// TIA Portal project "SiemensS7-modbus-TCPIP-server" (V16)

(* hardware
DEVICE "S71500/ET200MP station_1"  S7-1500 station
   slot 0: "Rail_0"  Rack  6ES7 590-1***0-0AA0
   slot 1: "PLC_1"  CPU 1512C-1 PN  6ES7 512-1CK01-0AB0  V2.8
      slot 3: "CPU display_1"  6ES7591-1AA00-0AA0
      slot 32768: "PROFINET interface_1"  X1
         slot 32769: "Port_1"  X1 P1
         slot 32770: "Port_2"  X1 P2
      slot 34817: "Virtual CP interface port_1"  Virtual CP interface port  Virtual CP interface port
*)

// ===== PLC "PLC_1"  CPU 1512C-1 PN =====

VAR_GLOBAL   // PLC tag table "Default tag table"
   "System_Byte" AT %MB1 : Byte;
   "FirstScan" AT %M1.0 : Bool;
   "DiagStatusUpdate" AT %M1.1 : Bool;
   "AlwaysTRUE" AT %M1.2 : Bool;
   "AlwaysFALSE" AT %M1.3 : Bool;
   "Clock_Byte" AT %MB0 : Byte;
   "Clock_10Hz" AT %M0.0 : Bool;
   "Clock_5Hz" AT %M0.1 : Bool;
   "Clock_2.5Hz" AT %M0.2 : Bool;
   "Clock_2Hz" AT %M0.3 : Bool;
   "Clock_1.25Hz" AT %M0.4 : Bool;
   "Clock_1Hz" AT %M0.5 : Bool;
   "Clock_0.625Hz" AT %M0.6 : Bool;
   "Clock_0.5Hz" AT %M0.7 : Bool;
   "Tag_1" AT %M1.4 : Bool;
END_VAR

DATA_BLOCK "Connect"   // DB1
{ S7_Optimized_Access := 'FALSE' }
VERSION : 0.1
   VAR
      Req : Bool := false;
      Disconnect : Bool;
      SND : TCON_IP_v4;
      RCV : TCON_IP_v4;
   END_VAR
BEGIN
   SND.InterfaceId := 64;
   SND.ID := 1;
   SND.ConnectionType := 11;
   SND.ActiveEstablished := True;
   SND.RemotePort := 502;
   SND.RemoteAddress.ADDR[1] := 192;
   SND.RemoteAddress.ADDR[2] := 168;
   SND.RemoteAddress.ADDR[3] := 0;
   SND.RemoteAddress.ADDR[4] := 114;
   RCV.InterfaceId := 64;
   RCV.ID := 2;
   RCV.ConnectionType := 11;
   RCV.ActiveEstablished := True;
   RCV.RemoteAddress.ADDR[1] := 192;
   RCV.RemoteAddress.ADDR[2] := 168;
   RCV.RemoteAddress.ADDR[3] := 0;
   RCV.RemoteAddress.ADDR[4] := 114;
   RCV.RemotePort := 502;
   SND.LocalPort := 0;
   RCV.LocalPort := 0;
END_DATA_BLOCK

DATA_BLOCK "Data"   // DB2
{ S7_Optimized_Access := 'FALSE' }
VERSION : 0.1
   VAR
      SND : Array[0..3] of Int;
      RCV : Array[0..1] of Int;
   END_VAR
BEGIN
   SND[0] := 0;
   SND[1] := 0;
   SND[2] := 0;
   SND[3] := 0;
END_DATA_BLOCK

DATA_BLOCK "Modbus_DB"   // DB3
{ S7_Optimized_Access := 'TRUE' }
VERSION : 0.1
// stored: InstanceOfName Modbus
"Modbus"
BEGIN
END_DATA_BLOCK

FUNCTION_BLOCK "Modbus"   // FB1, LAD
{ S7_Optimized_Access := 'TRUE' }
VERSION : 0.1
   VAR
      MB_CLIENT_Instance : MB_CLIENT;
      R_TRIG_Instance : R_TRIG;
      MB_CLIENT_Instance_1 : MB_CLIENT;
   END_VAR
BEGIN

REGION Network 1
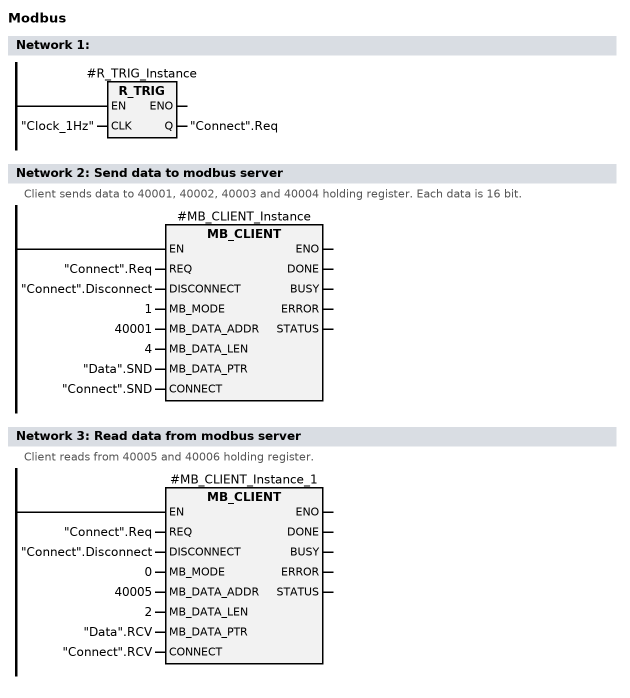
   #R_TRIG_Instance(CLK := "Clock_1Hz", Q => "Connect".Req);   // R_TRIG
END_REGION

REGION Network 2: Send data to modbus server
   // Client sends data to 40001, 40002, 40003 and 40004 holding register. Each data is 16 bit.
   #MB_CLIENT_Instance(REQ := "Connect".Req,   // MB_CLIENT
                       DISCONNECT := "Connect".Disconnect,
                       MB_MODE := 1,
                       MB_DATA_ADDR := 40001,
                       MB_DATA_LEN := 4,
                       MB_DATA_PTR := "Data".SND,
                       CONNECT := "Connect".SND);
END_REGION

REGION Network 3: Read data from modbus server
   // Client reads from 40005 and 40006 holding register.
   #MB_CLIENT_Instance_1(REQ := "Connect".Req,   // MB_CLIENT
                         DISCONNECT := "Connect".Disconnect,
                         MB_MODE := 0,
                         MB_DATA_ADDR := 40005,
                         MB_DATA_LEN := 2,
                         MB_DATA_PTR := "Data".RCV,
                         CONNECT := "Connect".RCV);
END_REGION
END_FUNCTION_BLOCK

ORGANIZATION_BLOCK "Main"   // OB1, LAD, ProgramCycle
TITLE = "Main Program Sweep (Cycle)"
{ S7_Optimized_Access := 'TRUE' }
VERSION : 0.1
   VAR_INPUT
      Initial_Call : Bool;   // Initial call of this OB
      Remanence : Bool;   // =True, if remanent data are available
   END_VAR
BEGIN

REGION Network 1
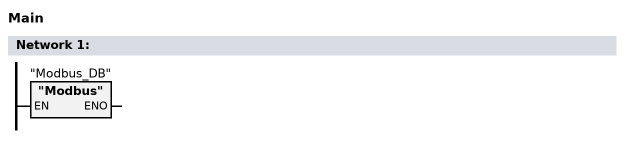
   RUNG wire#powerrail
      "Modbus_DB"()
   END_RUNG
   // the same network as SCL:
   "Modbus_DB"();   // "Modbus"
END_REGION
END_ORGANIZATION_BLOCK